Fanuc KAREL source: kb00131.KL

-- PROVISIONAL review KL for V770-1; original PC SHA256 3fa522feb5060dc4145719ef4dc61956c263cfa3cd4bbca7c9ec7b0b932b38a6
-- Incomplete behavior may be omitted. Consult companion uncertainty JSON. Do not deploy.
PROGRAM KB00131
%NOLOCKGROUP
BEGIN
  -- UNRESOLVED_PC offsets 5-14; opcodes 3F,75
  -- UNRESOLVED_PC offsets 19-26; opcodes 9D,23
  -- UNRESOLVED_PC offsets 31-38; opcodes 9D,23
  -- UNRESOLVED_PC offsets 43-50; opcodes 9D,23
  -- UNRESOLVED_PC offsets 55-64; opcodes 3F,75
  -- UNRESOLVED_PC offsets 69-76; opcodes 9D,23
  -- UNRESOLVED_PC offsets 81-88; opcodes 9D,23
  -- UNRESOLVED_PC offsets 93-143; opcodes 27,22,2A,22,22,22,22,2A,22,22,31
  -- UNRESOLVED_PC offsets 148-152; opcodes 7F
END KB00131
